Fanuc KAREL source: kt00962.KL

-- PROVISIONAL review KL for V1013-1; original PC SHA256 430097954dfac350a47f39d75140932b5bf0d864ef6dc92789df9871c9dacdc9
-- Incomplete behavior may be omitted. Consult companion uncertainty JSON. Do not deploy.
PROGRAM KT00962
%NOLOCKGROUP
VAR
  ENTRY : INTEGER
  PNAME : STRING[80]
  VNAME : STRING[80]
  STATUS : INTEGER
-- UNRESOLVED_DECL VALUE type=000101
BEGIN
  -- UNRESOLVED_PC offsets 5-12; opcodes 9C,23
  -- UNRESOLVED_PC offsets 17-25; opcodes 3F,75
  -- UNRESOLVED_PC offsets 30-43; opcodes 3F,75
  -- UNRESOLVED_PC offsets 48-92; opcodes 27,22,22,2A,22,2A,22,1C,22,B0
  -- UNRESOLVED_PC offsets 97-101; opcodes 7F
END KT00962
